// TIA Portal V17 export
// export: Created 2024-09-02T12:49:54.7886662Z, ExportSetting WithDefaults, DisplayName Totally Integrated Automation Portal, DisplayVersion V17, DisplayName TIA Portal Openness, DisplayVersion V17, DisplayName TIA Portal Version Control Interface, DisplayVersion V17, DisplayName STEP 7 Professional, DisplayVersion V17, DisplayName STEP 7 Safety, DisplayVersion V17, DisplayName WinCC Professional, DisplayVersion V17
FUNCTION "AnwFC_IBM_Mode" : Void   // FC0, LAD
TITLE = IBM Mode
{ S7_Optimized_Access := 'TRUE' }
AUTHOR : OlegFuehrus
VERSION : 0.1
// Motor potentiometer up / Nach IBM löschen
// stored: AutoNumber false, IsIECCheckEnabled false, SetENOAutomatically false, UDAEnableTagReadback false
   VAR_TEMP
      t_RET_VAL : Int;
      t_Date_and_Time : Date_And_Time;
      t_Ablage_Pos : Int;
      t_Prog_Nr : Int;
   END_VAR
BEGIN

REGION Network 1: IBS Fixed status "1" / IBS Fester Status "1"
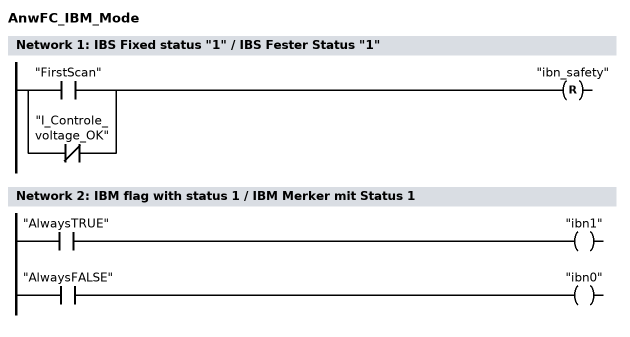
   RUNG wire#powerrail
      Contact( "FirstScan" )
      wire#w1
      R_Coil( "ibn_safety" )
   END_RUNG
   RUNG wire#powerrail
      I_Contact( "I_Controle_voltage_OK" )
   END_RUNG wire#w1
   // the same network as SCL:
   IF "FirstScan" OR NOT "I_Controle_voltage_OK" THEN "ibn_safety" := FALSE; END_IF;
END_REGION

REGION Network 2: IBM flag with status 1 / IBM Merker mit Status 1
   RUNG wire#powerrail
      Contact( "AlwaysTRUE" )
      Coil( "ibn1" )
   END_RUNG
   RUNG wire#powerrail
      Contact( "AlwaysFALSE" )
      Coil( "ibn0" )
   END_RUNG
   // the same network as SCL:
   "ibn1" := "AlwaysTRUE";
   "ibn0" := "AlwaysFALSE";
END_REGION
END_FUNCTION
